(* Logix 5000 project; controller WWTP_SOLIDS_CLX vendor 1 type 14 code 54 rev 17.2; software revision 17.00; part 3 of 16 *)
(* tags used below, declared in another part *)
   Inp : BOOL;   // Alarm Condition Input 1=Alarm
   Cfg_ResetReqd : BOOL;   // 1=Reset required to clear Alarm
   Cfg_AckReqd : BOOL;   // 1=Acknowledge required for Alarm
   Cfg_Severity : SINT;   // 1=Info Only; 2=Warning; 3=Process Exception; 4=Fault
   Cfg_MinDuration : DINT;   // Minimum time (sec) Input must stay on to generate Alarm
   PCmd_Ack : BOOL;   // Program Command to Acknowledge alarm
   PCmd_Inhibit : BOOL;   // Program Command to Inhibit alarm (force Alm to 0)
   PCmd_Uninhibit : BOOL;   // Program Command to Uninhibit alarm
   OCmd_Ack : BOOL;   // Operator Command to Acknowledge alarm
   OCmd_Disable : BOOL;   // Operator Command to Disable alarm (force Alm to 0)
   OCmd_Enable : BOOL;   // Operator Command to Enable alarm
   Alm : BOOL;   // Alarm output 1=In Alarm
   Ack : BOOL;   // Alarm acknowledged status: 1=Ack rcvd
   Disabled : BOOL;   // 1=Alarm has been Disabled by Operator (will not be sent)
   Inhibited : BOOL;   // 1=Alarm has been Inhibited by logic (will not be sent)
   Suppressed : BOOL;   // 1=Alarm has been suppressed (not visible on HMI)
   Rdy_Disable : BOOL;   // Ready to receive OCmd_Disable (enable button)
(* P_Alarm, continued *)

ROUTINE Prescan   (* ladder *)
// Clear "lurking" Commands
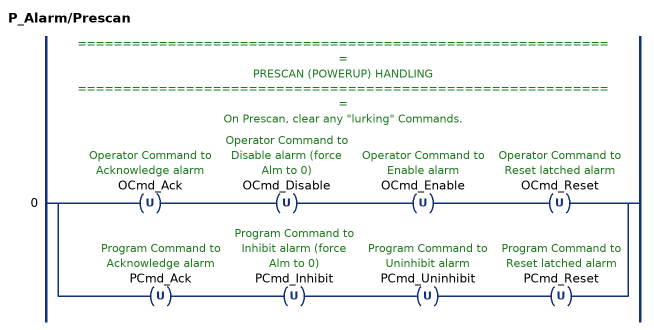
   // ============================================================
   // PRESCAN (POWERUP) HANDLING
   // ============================================================
   // On Prescan, clear any "lurking" Commands.
   0: [OTU(OCmd_Ack) OTU(OCmd_Disable) OTU(OCmd_Enable) OTU(OCmd_Reset) ,OTU(PCmd_Ack) OTU(PCmd_Inhibit) OTU(PCmd_Uninhibit) OTU(PCmd_Reset) ];
END_ROUTINE
END_ADD_ON_INSTRUCTION

ADD_ON_INSTRUCTION P_DIn   (* revision 0.29, ExecutePrescan, ExecuteEnableInFalse *)
// Discrete Input
// Revision note:
// Aligned name, description and local STRING values, sizes, across instructions.
// Help:
// This instruction monitors a discrete (1 / 0) input and checks for alarm conditions.
// The Inp_Gate input must be set (=1, its default value) and the alarm enabled for
// the alarm (Alm) to occur.  The alarm will not occur until the Inp_Gate input has
// been set for the Gate Delay (Cfg_GateDly) time.  The Gate is used to enable the
// alarm when some other condition is true; for example, a high vibration switch should
// only generate an alarm when the associated motor has been running long enough
// to stabilize.
// The alarm is generated when the Inp_PV (process variable) input is different from
// the Inp_Target (target) input.  The Target indicates the "normal" condition.  For
// example, a flow switch should indicate flow when a pump is running and should
// not indicate flow when a pump is stopped.  The pump run status is used as the
// Target input, and when the switch does not match the target (within the allotted
// time), the Alarm (Flow Loss / Switch Failure) is generated.
// NOTE: the Inp_PV is inverted when the rung condition is false -- this allows the
// input to be a condition on the rung with P_DIn rather than mapped into Inp_PV.
// See P_DIn documentation for details.
// This instruction includes a substitute PV capability for a manually-entered state.
// This may be useful when a sensor is out for repair or for simulation and testing.
VAR_INPUT
   Inp_PV : BOOL := 1; {visible}   // Input Signal (process variable) from Sensor
   Inp_PVBad : BOOL;   // Input Comm Status or Quality 1=Bad, 0=OK
   Inp_Target : BOOL := 1; {visible}   // Target State of Input (Alarm if not in Target State)
   Inp_Gate : BOOL := 1; {visible}   // Gate Condition (=1 to enable Alarm)
   Inp_Sim : BOOL;   // 1=Use simulated PV (Set_SimPV); 0=Use Input (Inp_PV)
   Inp_Reset : BOOL;   // 1=Reset Alarm requiring reset
   Cfg_NoSubstPV : BOOL;   // 1=Disallow selection of Substitute PV
   Cfg_NormTextVis : BOOL := 1;   // 1=Display state text in "normal" state (= target), 0=hide (some HMI objects)
   Cfg_PCmdClear : BOOL := 1;   // 1=Clear Program Commands on receipt 0=Leave Set
   Cfg_HasTgtDisagreeAlm : BOOL;   // 1=Target Disagree Alarm exists and will be checked
   Cfg_TgtDisagreeResetReqd : BOOL;   // 1=Target Disagree Alarm is latched in, requires Reset Command to clear
   Cfg_TgtDisagreeAckReqd : BOOL := 1;   // 1=Target Disagree Alarm must be acknowledged
   Cfg_TgtDisagreeSeverity : SINT := 3;   // Target Disagree Alarm Severity: 1=info, 2=warn, 3=excep, 4=fault
   Cfg_GateDly : DINT;   // Time Inp_Gate must be true before Alarm is checked (sec)
   Cfg_Debounce : REAL;   // Minimum time Status must maintain state, (sec)
   Cfg_TgtDisagreeMinDuration : DINT;   // Minimum time Input must disagree with target to generate an Alarm (sec)
   MSet_SubstPV : BOOL;   // Maintenance-Entered Substitute PV
   Set_SimPV : BOOL;   // PV used in Simulation (Inp_Sim=1)
   PCmd_Reset : BOOL;   // Program Command to Reset all latched Alarms
   PCmd_TgtDisagreeAck : BOOL;   // Program Command to Acknowledge the Target Disagree Alarm
   PCmd_TgtDisagreeInhibit : BOOL;   // Program Command to Inhibit the Target Disagree Alarm
   PCmd_TgtDisagreeUninhibit : BOOL;   // Program Command to Uninhibit the Target Disagree Alarm
   MCmd_SubstPV : BOOL;   // Maintenance Command to use Substitute PV (override input)
   MCmd_InpPV : BOOL;   // Maintenance Command to use Input PV (normal)
   OCmd_Reset : BOOL;   // Operator Command to Reset all latched Alarms
END_VAR
VAR_OUTPUT
   Val_Notify : SINT;   // Current Alarm Level and Acknowledgement (enumeration)
   Sts : BOOL; {visible}   // Discrete Input Status (incl. Debounce, Manual Override, if used)
   Sts_PV : BOOL; {visible}   // Discrete Input Status (actual, not subject to Override)
   Sts_SubstPV : BOOL;   // 1=Using Substitute PV (Input being overridden)
   Sts_InpPV : BOOL;   // 1=Using Input PV (normal)
   Sts_PVBad : BOOL;   // Input Comm Status/ Quality (0=OK, 1=Bad)
   Sts_Err : BOOL; {visible}   // 1=Error in Config: see detail bits for reason
   Err_Timer : BOOL;   // 1=Error in Config: Invalid Timer Preset (use 0 to 2147483)
   Err_Alarm : BOOL;   // 1=Error in Config: Invalid Alarm Min Duration or Severity
   Sts_TgtDisagree : BOOL;   // 1=Input is not in Target state
   Alm_TgtDisagree : BOOL;   // 1=Alarm: Input is not in Target state
   Ack_TgtDisagree : BOOL;   // 1=Target Disagree Alarm has been acknowledged
   Sts_TgtDisagreeDisabled : BOOL;   // 1=Target Disagree Alarm is Disabled (not saved or sent)
   Sts_TgtDisagreeInhibited : BOOL;   // 1=Target Disagree Alarm is Inhibited by logic
   Sts_TgtDisagreeSuppressed : BOOL;   // 1=Target Disagree Alarm is Suppressed (logged only)
   Rdy_SubstPV : BOOL;   // 1=Ready for MCmd_SubstPV
   Rdy_InpPV : BOOL;   // 1=Ready for MCmd_InpPV
   Rdy_Reset : BOOL;   // 1=Ready for Operator Alarm Reset Command
END_VAR
VAR
   Wrk_GateDlyT : TIMER;   // Gate Delay timer
   Cfg_Tag : STRING_20 := 'P_DIn';   // Tagname for display on HMI
   Cfg_Desc : STRING_40 := 'Discrete Input';   // Description for display on HMI
   Cfg_Label : STRING_20 := 'Discrete Input';   // Label for graphic symbol displayed on HMI
   Wrk_Sts : BOOL;   // Internal Status (after Manual Override selection)
   TgtDisagree : P_Alarm := (Inp := 1, Cfg_AckReqd := 1, Cfg_Severity := 3, Ack := 1, Rdy_Disable := 1);   // Target Disagree Alarm
   Wrk_FallT : TIMER;   // Timer to ensure Status LOW time on falling edge
   Wrk_RiseT : TIMER;   // Timer to ensure Status HIGH time on rising edge
   Wrk_SubstPV : BOOL;   // Internal flag: Using Substitute PV
   Cfg_1StText : STRING_8 := 'On';   // Text to display in PV=1 State
   Cfg_0StText : STRING_8 := 'Off';   // Text to display in PV=0 State
END_VAR

ROUTINE EnableInFalse   (* ladder *)
// Inverts Inp_PV to allow mapping input using XIC/XIO on rung
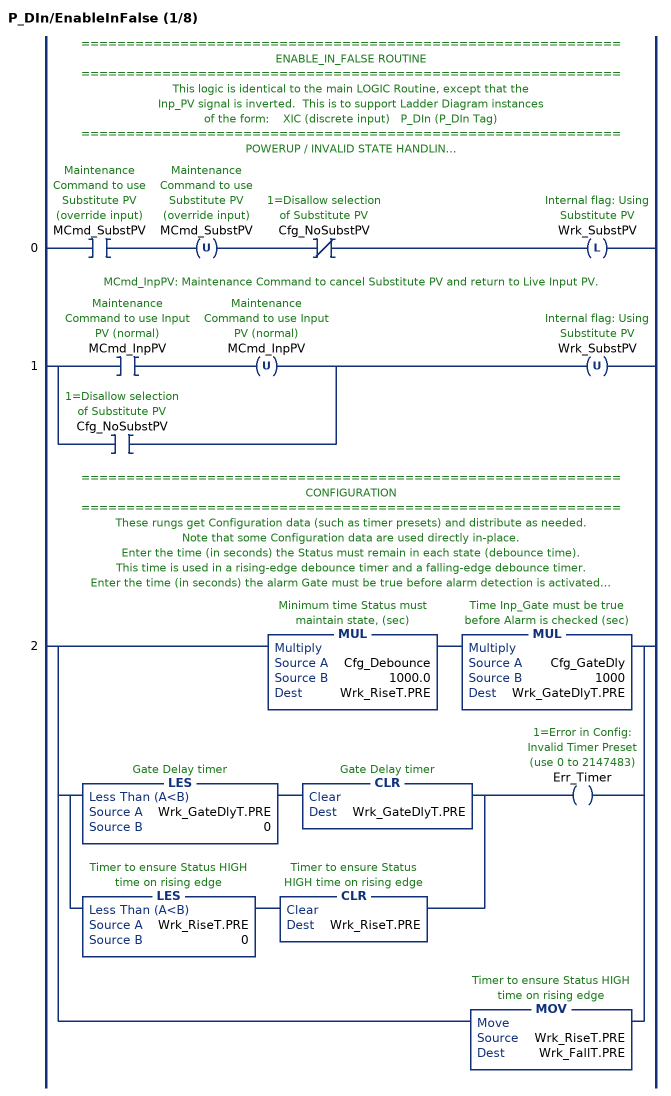
   // ============================================================
   // ENABLE_IN_FALSE ROUTINE
   // ============================================================
   // This logic is identical to the main LOGIC Routine, except that the
   // Inp_PV signal is inverted.  This is to support Ladder Diagram instances
   // of the form:    XIC (discrete input)   P_DIn (P_DIn Tag)
   // ============================================================
   // POWERUP / INVALID STATE HANDLING
   // ============================================================
   // All internal Work (state) bits maintain states through a power cycle and are
   // independent.  No Powerup / Invalid State Handling logic is required.
   // ============================================================
   // COMMAND PROCESSING
   // ============================================================
   // These rungs handle received Commands:
   // NOTE:  Operator Commands for P_Alarm are sent directly to the contained P_Alarm AOI.
   // MCmd_SubstPV: Maintenance Command to select Maintenance-entered substitute PV
   // Do not allow this Commands if Cfg_NoSubstPV is set.
   0: XIC(MCmd_SubstPV)OTU(MCmd_SubstPV)XIO(Cfg_NoSubstPV)OTL(Wrk_SubstPV);
   // MCmd_InpPV: Maintenance Command to cancel Substitute PV and return to Live Input PV.
   1: [XIC(MCmd_InpPV) OTU(MCmd_InpPV) ,XIC(Cfg_NoSubstPV) ]OTU(Wrk_SubstPV);
   // ============================================================
   // CONFIGURATION
   // ============================================================
   // These rungs get Configuration data (such as timer presets) and distribute as needed.
   // Note that some Configuration data are used directly in-place.
   // Enter the time (in seconds) the Status must remain in each state (debounce time).
   // This time is used in a rising-edge debounce timer and a falling-edge debounce timer.
   // Enter the time (in seconds) the alarm Gate must be true before alarm detection is activated.
   // If the timer preset calcuated wraps negative (more than 2.14... million seconds), then establish
   // a valid limit value for the Preset.  Note that a negative timer preset will fault the controller!!!
   2: [MUL(Cfg_Debounce,1000.0,Wrk_RiseT.PRE) MUL(Cfg_GateDly,1000,Wrk_GateDlyT.PRE) ,[LES(Wrk_GateDlyT.PRE,0) CLR(Wrk_GateDlyT.PRE) ,LES(Wrk_RiseT.PRE,0) CLR(Wrk_RiseT.PRE) ] OTE(Err_Timer) ,MOV(Wrk_RiseT.PRE,Wrk_FallT.PRE) ];
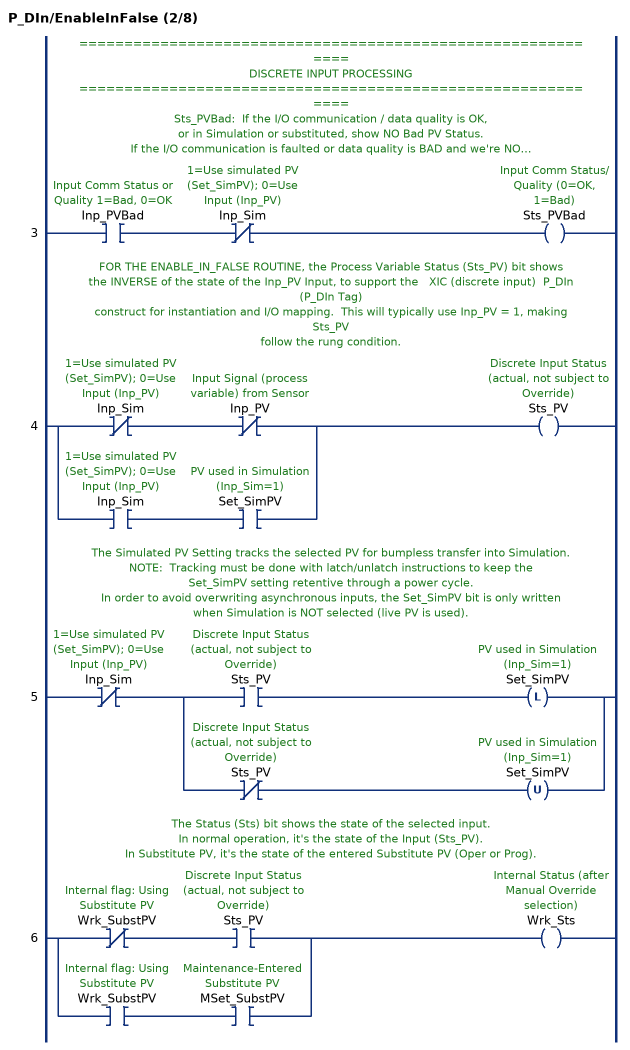
   // ============================================================
   // DISCRETE INPUT PROCESSING
   // ============================================================
   // Sts_PVBad:  If the I/O communication / data quality is OK,
   // or in Simulation or substituted, show NO Bad PV Status.
   // If the I/O communication is faulted or data quality is BAD and we're NOT
   // in Simulation or using substitute PV, show the Bad PV Status.
   3: XIC(Inp_PVBad)XIO(Inp_Sim)OTE(Sts_PVBad);
   // FOR THE ENABLE_IN_FALSE ROUTINE, the Process Variable Status (Sts_PV) bit shows
   // the INVERSE of the state of the Inp_PV Input, to support the   XIC (discrete input)  P_DIn (P_DIn Tag)
   // construct for instantiation and I/O mapping.  This will typically use Inp_PV = 1, making Sts_PV
   // follow the rung condition.
   4: [XIO(Inp_Sim) XIO(Inp_PV) ,XIC(Inp_Sim) XIC(Set_SimPV) ]OTE(Sts_PV);
   // The Simulated PV Setting tracks the selected PV for bumpless transfer into Simulation.
   // NOTE:  Tracking must be done with latch/unlatch instructions to keep the
   // Set_SimPV setting retentive through a power cycle.
   // In order to avoid overwriting asynchronous inputs, the Set_SimPV bit is only written
   // when Simulation is NOT selected (live PV is used).
   5: XIO(Inp_Sim)[XIC(Sts_PV) OTL(Set_SimPV) ,XIO(Sts_PV) OTU(Set_SimPV) ];
   // The Status (Sts) bit shows the state of the selected input.
   // In normal operation, it's the state of the Input (Sts_PV).
   // In Substitute PV, it's the state of the entered Substitute PV (Oper or Prog).
   6: [XIO(Wrk_SubstPV) XIC(Sts_PV) ,XIC(Wrk_SubstPV) XIC(MSet_SubstPV) ]OTE(Wrk_Sts);
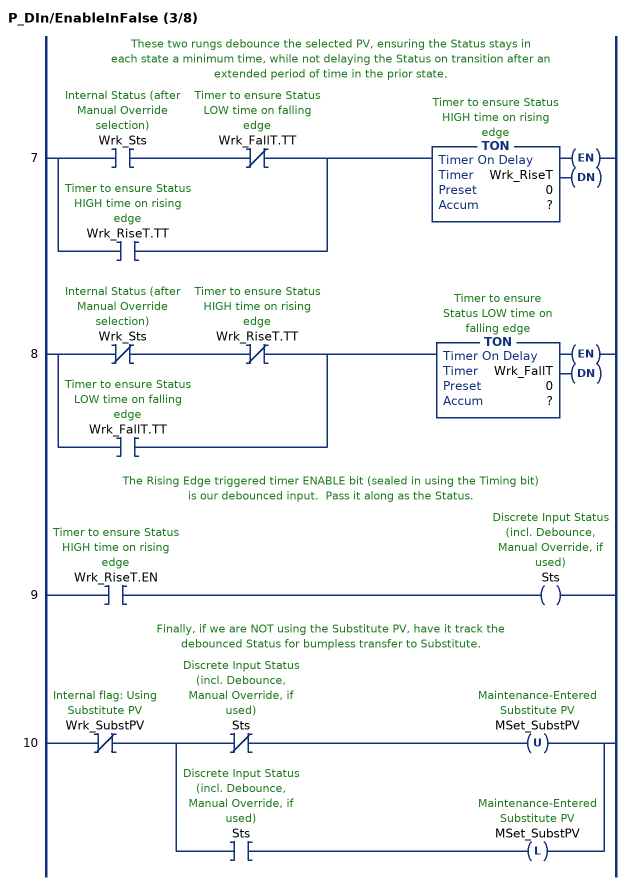
   // These two rungs debounce the selected PV, ensuring the Status stays in
   // each state a minimum time, while not delaying the Status on transition after an
   // extended period of time in the prior state.
   7: [XIC(Wrk_Sts) XIO(Wrk_FallT.TT) ,XIC(Wrk_RiseT.TT) ]TON(Wrk_RiseT,?,?);
   8: [XIO(Wrk_Sts) XIO(Wrk_RiseT.TT) ,XIC(Wrk_FallT.TT) ]TON(Wrk_FallT,?,?);
   // The Rising Edge triggered timer ENABLE bit (sealed in using the Timing bit)
   // is our debounced input.  Pass it along as the Status.
   9: XIC(Wrk_RiseT.EN)OTE(Sts);
   // Finally, if we are NOT using the Substitute PV, have it track the
   // debounced Status for bumpless transfer to Substitute.
   10: XIO(Wrk_SubstPV)[XIO(Sts) OTU(MSet_SubstPV) ,XIC(Sts) OTL(MSet_SubstPV) ];
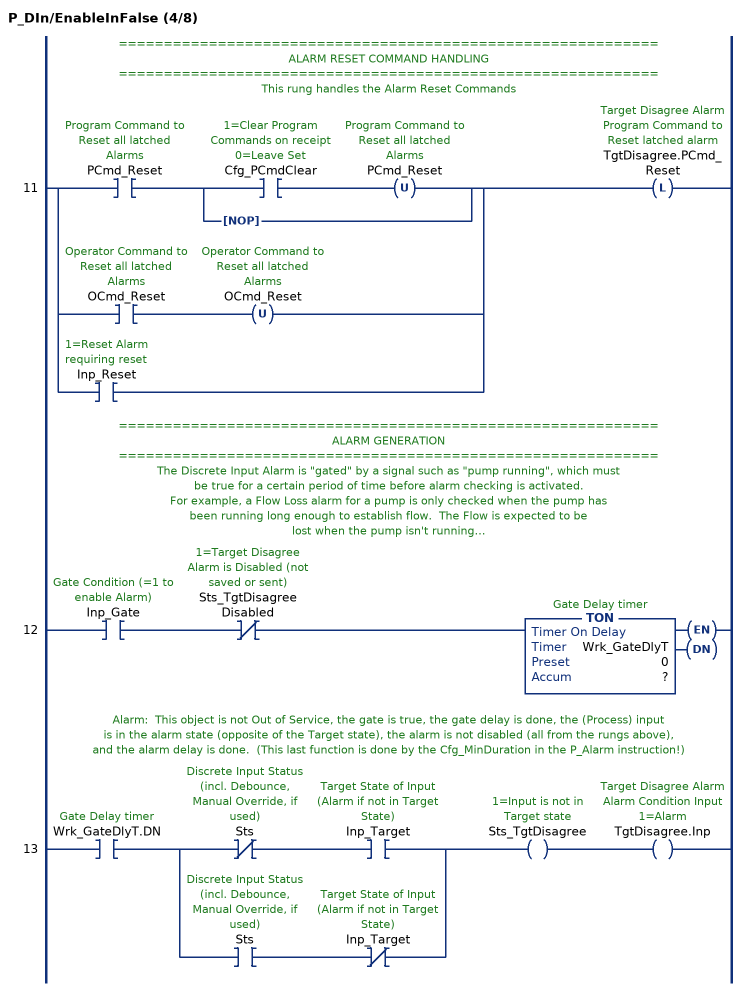
   // ============================================================
   // ALARM RESET COMMAND HANDLING
   // ============================================================
   // This rung handles the Alarm Reset Commands
   11: [XIC(PCmd_Reset) [XIC(Cfg_PCmdClear) OTU(PCmd_Reset) ,NOP() ] ,XIC(OCmd_Reset) OTU(OCmd_Reset) ,XIC(Inp_Reset) ]OTL(TgtDisagree.PCmd_Reset);
   // ============================================================
   // ALARM GENERATION
   // ============================================================
   // The Discrete Input Alarm is "gated" by a signal such as "pump running", which must
   // be true for a certain period of time before alarm checking is activated.
   // For example, a Flow Loss alarm for a pump is only checked when the pump has
   // been running long enough to establish flow.  The Flow is expected to be
   // lost when the pump isn't running!
   // If no gating signal is available, set Inp_Gate to 1 and Cfg_GateT to 0.
   12: XIC(Inp_Gate)XIO(Sts_TgtDisagreeDisabled)TON(Wrk_GateDlyT,?,?);
   // Alarm:  This object is not Out of Service, the gate is true, the gate delay is done, the (Process) input
   // is in the alarm state (opposite of the Target state), the alarm is not disabled (all from the rungs above),
   // and the alarm delay is done.  (This last function is done by the Cfg_MinDuration in the P_Alarm instruction!)
   13: XIC(Wrk_GateDlyT.DN)[XIO(Sts) XIC(Inp_Target) ,XIC(Sts) XIO(Inp_Target) ]OTE(Sts_TgtDisagree)OTE(TgtDisagree.Inp);
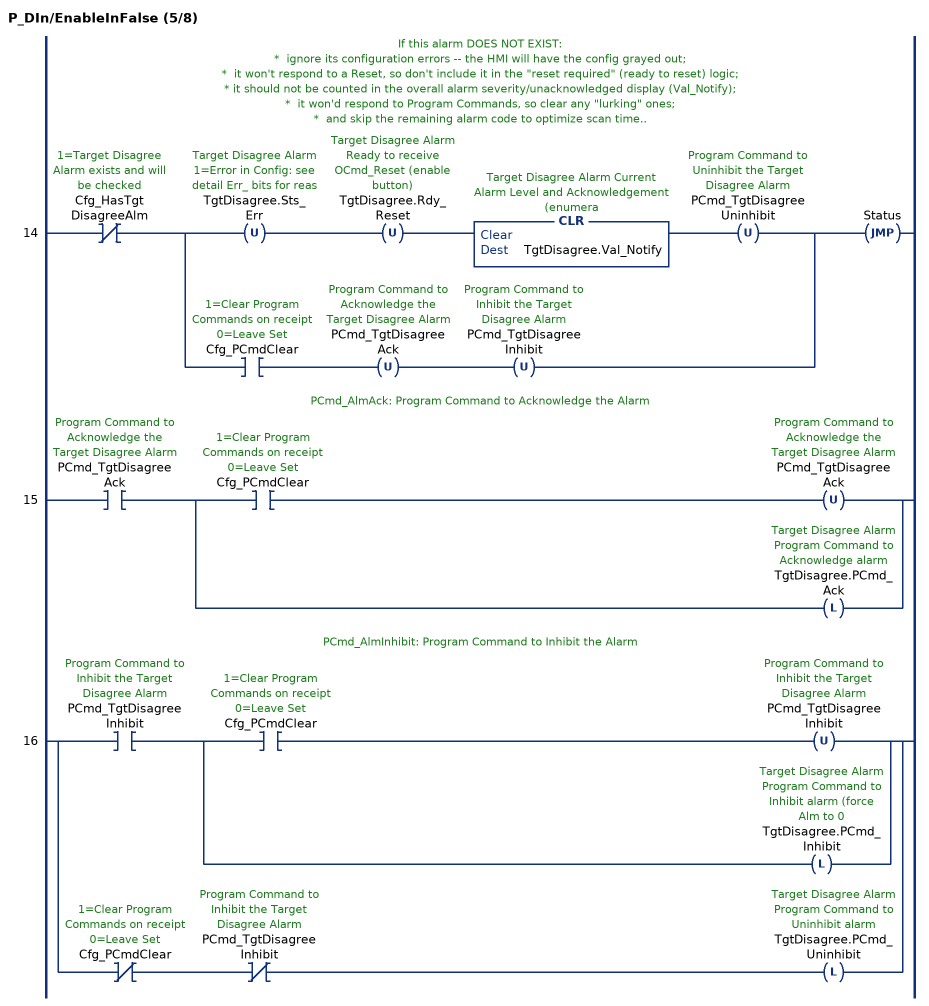
   // If this alarm DOES NOT EXIST:
   // *  ignore its configuration errors -- the HMI will have the config grayed out;
   // *  it won't respond to a Reset, so don't include it in the "reset required" (ready to reset) logic;
   // * it should not be counted in the overall alarm severity/unacknowledged display (Val_Notify);
   // *  it won'd respond to Program Commands, so clear any "lurking" ones;
   // *  and skip the remaining alarm code to optimize scan time..
   14: XIO(Cfg_HasTgtDisagreeAlm)[OTU(TgtDisagree.Sts_Err) OTU(TgtDisagree.Rdy_Reset) CLR(TgtDisagree.Val_Notify) OTU(PCmd_TgtDisagreeUninhibit) ,XIC(Cfg_PCmdClear) OTU(PCmd_TgtDisagreeAck) OTU(PCmd_TgtDisagreeInhibit) ]JMP(Status);
   // PCmd_AlmAck: Program Command to Acknowledge the Alarm
   15: XIC(PCmd_TgtDisagreeAck)[XIC(Cfg_PCmdClear) OTU(PCmd_TgtDisagreeAck) ,OTL(TgtDisagree.PCmd_Ack) ];
   // PCmd_AlmInhibit: Program Command to Inhibit the Alarm
   16: [XIC(PCmd_TgtDisagreeInhibit) [XIC(Cfg_PCmdClear) OTU(PCmd_TgtDisagreeInhibit) ,OTL(TgtDisagree.PCmd_Inhibit) ] ,XIO(Cfg_PCmdClear) XIO(PCmd_TgtDisagreeInhibit) OTL(TgtDisagree.PCmd_Uninhibit) ];
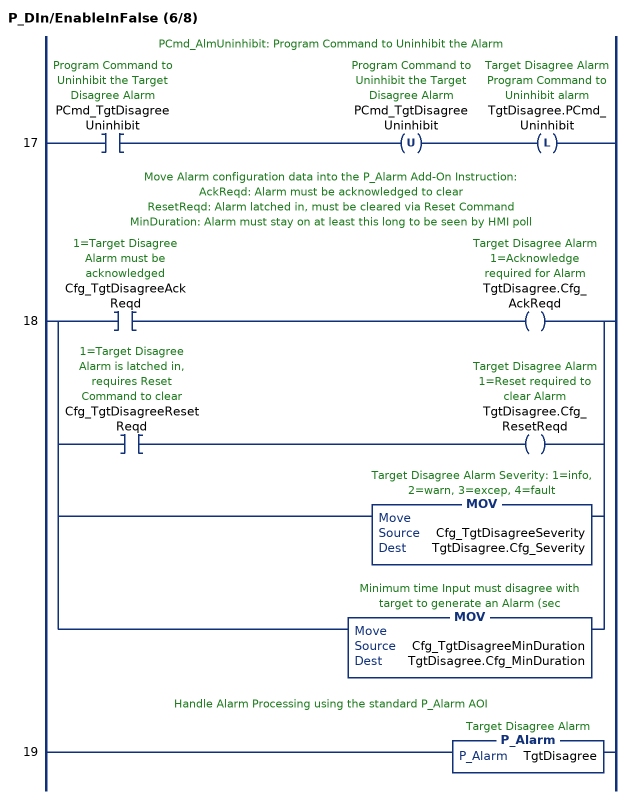
   // PCmd_AlmUninhibit: Program Command to Uninhibit the Alarm
   17: XIC(PCmd_TgtDisagreeUninhibit)OTU(PCmd_TgtDisagreeUninhibit)OTL(TgtDisagree.PCmd_Uninhibit);
   // Move Alarm configuration data into the P_Alarm Add-On Instruction:
   // AckReqd: Alarm must be acknowledged to clear
   // ResetReqd: Alarm latched in, must be cleared via Reset Command
   // MinDuration: Alarm must stay on at least this long to be seen by HMI poll
   18: [XIC(Cfg_TgtDisagreeAckReqd) OTE(TgtDisagree.Cfg_AckReqd) ,XIC(Cfg_TgtDisagreeResetReqd) OTE(TgtDisagree.Cfg_ResetReqd) ,MOV(Cfg_TgtDisagreeSeverity,TgtDisagree.Cfg_Severity) ,MOV(Cfg_TgtDisagreeMinDuration,TgtDisagree.Cfg_MinDuration) ];
   // Handle Alarm Processing using the standard P_Alarm AOI
   19: P_Alarm(TgtDisagree);
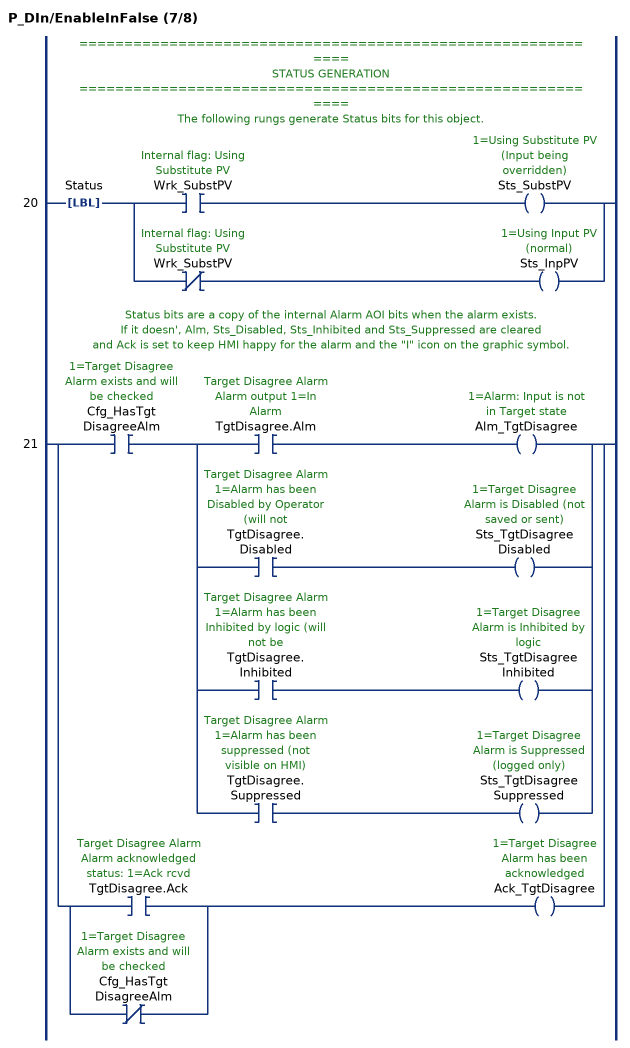
   // ============================================================
   // STATUS GENERATION
   // ============================================================
   // The following rungs generate Status bits for this object.
   20: LBL(Status)[XIC(Wrk_SubstPV) OTE(Sts_SubstPV) ,XIO(Wrk_SubstPV) OTE(Sts_InpPV) ];
   // Status bits are a copy of the internal Alarm AOI bits when the alarm exists.
   // If it doesn', Alm, Sts_Disabled, Sts_Inhibited and Sts_Suppressed are cleared
   // and Ack is set to keep HMI happy for the alarm and the "I" icon on the graphic symbol.
   21: [XIC(Cfg_HasTgtDisagreeAlm) [XIC(TgtDisagree.Alm) OTE(Alm_TgtDisagree) ,XIC(TgtDisagree.Disabled) OTE(Sts_TgtDisagreeDisabled) ,XIC(TgtDisagree.Inhibited) OTE(Sts_TgtDisagreeInhibited) ,XIC(TgtDisagree.Suppressed) OTE(Sts_TgtDisagreeSuppressed) ] ,[XIC(TgtDisagree.Ack) ,XIO(Cfg_HasTgtDisagreeAlm) ] OTE(Ack_TgtDisagree) ];
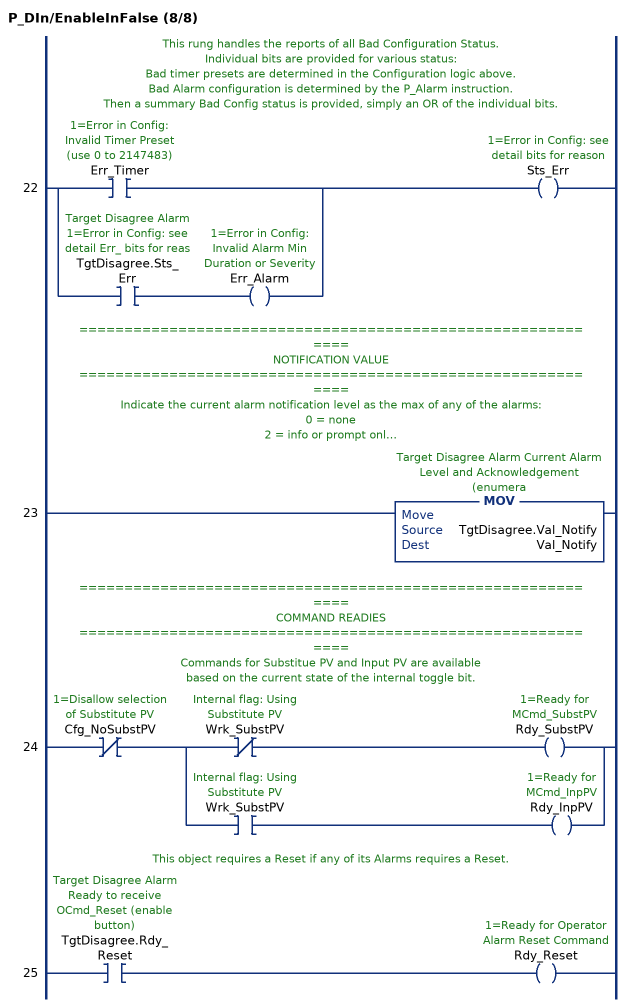
   // This rung handles the reports of all Bad Configuration Status.
   // Individual bits are provided for various status:
   // Bad timer presets are determined in the Configuration logic above.
   // Bad Alarm configuration is determined by the P_Alarm instruction.
   // Then a summary Bad Config status is provided, simply an OR of the individual bits.
   22: [XIC(Err_Timer) ,XIC(TgtDisagree.Sts_Err) OTE(Err_Alarm) ]OTE(Sts_Err);
   // ============================================================
   // NOTIFICATION VALUE
   // ============================================================
   // Indicate the current alarm notification level as the max of any of the alarms:
   // 0 = none
   // 2 = info or prompt only
   // 4 = warning
   // 6 = exception (equipment impact)
   // 8 = fault (equipment failure)
   // Add one for any unsuppressed alarm that is not acknowledged (for blink).
   23: MOV(TgtDisagree.Val_Notify,Val_Notify);
   // ============================================================
   // COMMAND READIES
   // ============================================================
   // Commands for Substitue PV and Input PV are available
   // based on the current state of the internal toggle bit.
   24: XIO(Cfg_NoSubstPV)[XIO(Wrk_SubstPV) OTE(Rdy_SubstPV) ,XIC(Wrk_SubstPV) OTE(Rdy_InpPV) ];
   // This object requires a Reset if any of its Alarms requires a Reset.
   25: XIC(TgtDisagree.Rdy_Reset)OTE(Rdy_Reset);
END_ROUTINE

ROUTINE Logic   (* ladder *)
// Normal Scan - status is updated and alarms are generated
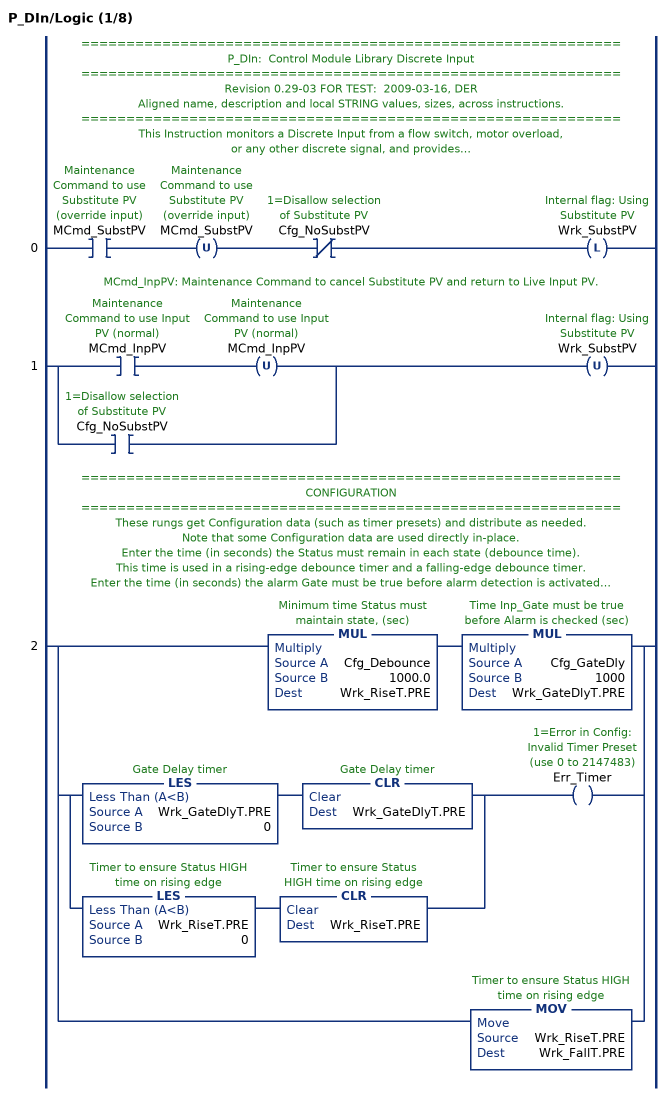
   // ============================================================
   // P_DIn:  Control Module Library Discrete Input
   // ============================================================
   // Revision 0.29-03 FOR TEST:  2009-03-16, DER
   // Aligned name, description and local STRING values, sizes, across instructions.
   // ============================================================
   // This Instruction monitors a Discrete Input from a flow switch, motor overload,
   // or any other discrete signal, and provides:
   // *  Status, with configurable names for the 0- and 1-states
   // *  An Alarm "Gate" signal (with delay), used to enable an Alarm under appropriate process conditions
   // *  A "Target" input -- the Alarm is raised when the input is not in the same
   // state as the Target for a configurable period of time
   // * Input debounce for both the rising and falling transitions
   // * Commands to inhibit or enable alarms
   // * Monitoring of input communication status
   // * Setting of a simulated input signal for process simulation
   // * Selection of Substitute PV (by Maintenance personnel) or normal PV
   // ============================================================
   // POWERUP / INVALID STATE HANDLING
   // ============================================================
   // All internal Work (state) bits maintain states through a power cycle and are
   // independent.  No Powerup / Invalid State Handling logic is required.
   // ============================================================
   // COMMAND PROCESSING
   // ============================================================
   // These rungs handle received Commands:
   // NOTE:  Operator Commands for P_Alarm are sent directly to the contained AOI.
   // MCmd_SubstPV: Maintenance Command to select Maintenance-entered substitute PV
   // Do not allow this Commands if Cfg_NoSubstPV is set.
   0: XIC(MCmd_SubstPV)OTU(MCmd_SubstPV)XIO(Cfg_NoSubstPV)OTL(Wrk_SubstPV);
   // MCmd_InpPV: Maintenance Command to cancel Substitute PV and return to Live Input PV.
   1: [XIC(MCmd_InpPV) OTU(MCmd_InpPV) ,XIC(Cfg_NoSubstPV) ]OTU(Wrk_SubstPV);
   // ============================================================
   // CONFIGURATION
   // ============================================================
   // These rungs get Configuration data (such as timer presets) and distribute as needed.
   // Note that some Configuration data are used directly in-place.
   // Enter the time (in seconds) the Status must remain in each state (debounce time).
   // This time is used in a rising-edge debounce timer and a falling-edge debounce timer.
   // Enter the time (in seconds) the alarm Gate must be true before alarm detection is activated.
   // If the timer preset calcuated wraps negative (more than 2.14... million seconds), then establish
   // a valid limit value for the Preset.  Note that a negative timer preset will fault the controller!!!
   2: [MUL(Cfg_Debounce,1000.0,Wrk_RiseT.PRE) MUL(Cfg_GateDly,1000,Wrk_GateDlyT.PRE) ,[LES(Wrk_GateDlyT.PRE,0) CLR(Wrk_GateDlyT.PRE) ,LES(Wrk_RiseT.PRE,0) CLR(Wrk_RiseT.PRE) ] OTE(Err_Timer) ,MOV(Wrk_RiseT.PRE,Wrk_FallT.PRE) ];
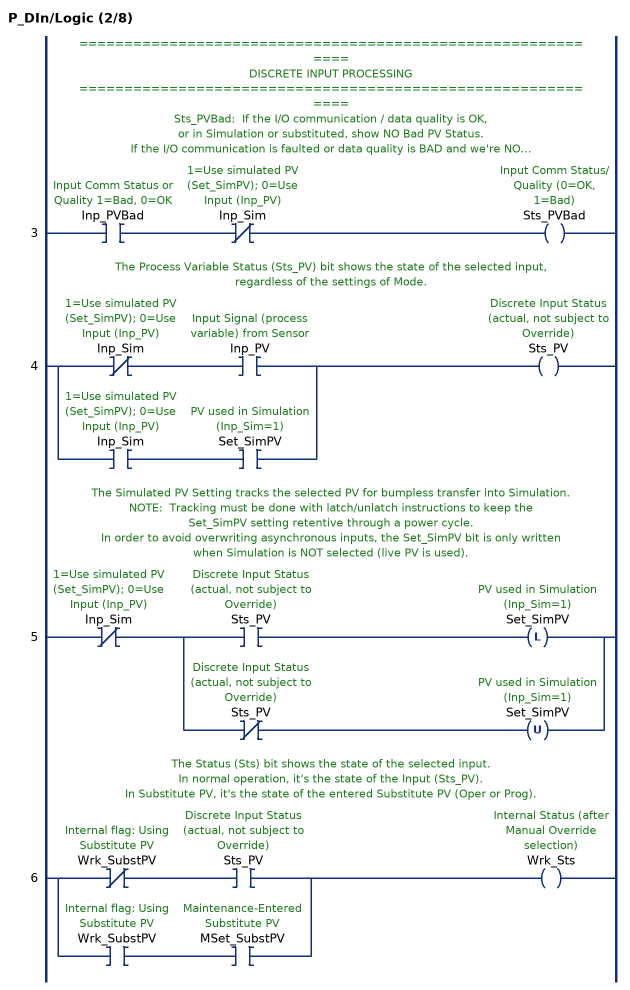
   // ============================================================
   // DISCRETE INPUT PROCESSING
   // ============================================================
   // Sts_PVBad:  If the I/O communication / data quality is OK,
   // or in Simulation or substituted, show NO Bad PV Status.
   // If the I/O communication is faulted or data quality is BAD and we're NOT
   // in Simulation or using substitute PV, show the Bad PV Status.
   3: XIC(Inp_PVBad)XIO(Inp_Sim)OTE(Sts_PVBad);
   // The Process Variable Status (Sts_PV) bit shows the state of the selected input,
   // regardless of the settings of Mode.
   4: [XIO(Inp_Sim) XIC(Inp_PV) ,XIC(Inp_Sim) XIC(Set_SimPV) ]OTE(Sts_PV);
   // The Simulated PV Setting tracks the selected PV for bumpless transfer into Simulation.
   // NOTE:  Tracking must be done with latch/unlatch instructions to keep the
   // Set_SimPV setting retentive through a power cycle.
   // In order to avoid overwriting asynchronous inputs, the Set_SimPV bit is only written
   // when Simulation is NOT selected (live PV is used).
   5: XIO(Inp_Sim)[XIC(Sts_PV) OTL(Set_SimPV) ,XIO(Sts_PV) OTU(Set_SimPV) ];
   // The Status (Sts) bit shows the state of the selected input.
   // In normal operation, it's the state of the Input (Sts_PV).
   // In Substitute PV, it's the state of the entered Substitute PV (Oper or Prog).
   6: [XIO(Wrk_SubstPV) XIC(Sts_PV) ,XIC(Wrk_SubstPV) XIC(MSet_SubstPV) ]OTE(Wrk_Sts);
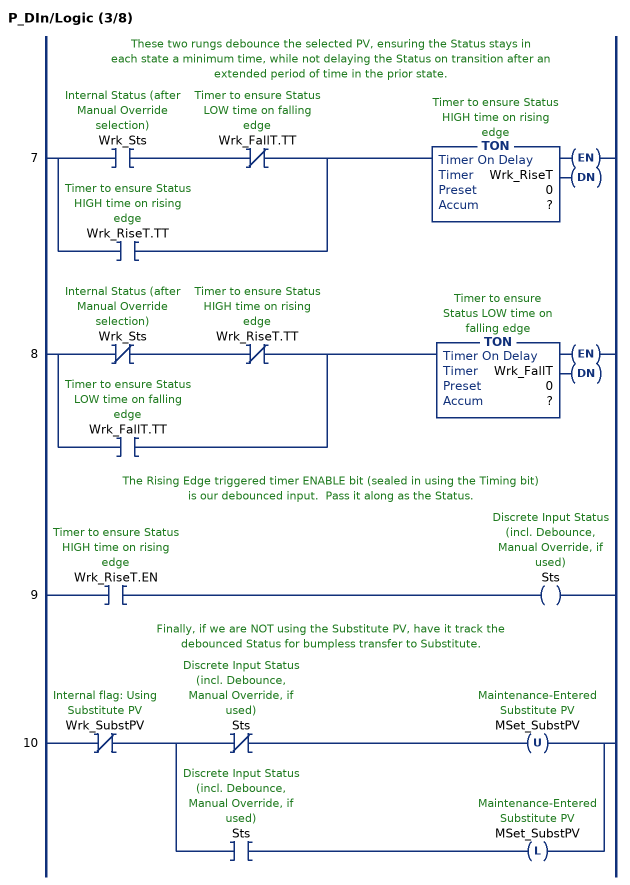
   // These two rungs debounce the selected PV, ensuring the Status stays in
   // each state a minimum time, while not delaying the Status on transition after an
   // extended period of time in the prior state.
   7: [XIC(Wrk_Sts) XIO(Wrk_FallT.TT) ,XIC(Wrk_RiseT.TT) ]TON(Wrk_RiseT,?,?);
   8: [XIO(Wrk_Sts) XIO(Wrk_RiseT.TT) ,XIC(Wrk_FallT.TT) ]TON(Wrk_FallT,?,?);
   // The Rising Edge triggered timer ENABLE bit (sealed in using the Timing bit)
   // is our debounced input.  Pass it along as the Status.
   9: XIC(Wrk_RiseT.EN)OTE(Sts);
   // Finally, if we are NOT using the Substitute PV, have it track the
   // debounced Status for bumpless transfer to Substitute.
   10: XIO(Wrk_SubstPV)[XIO(Sts) OTU(MSet_SubstPV) ,XIC(Sts) OTL(MSet_SubstPV) ];
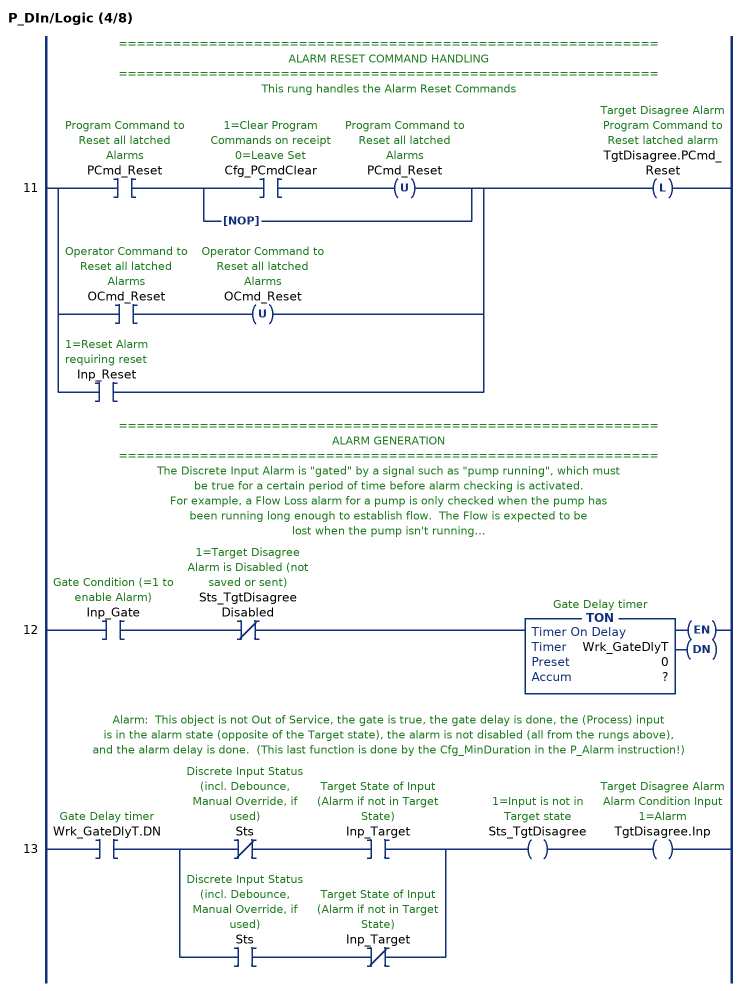
   // ============================================================
   // ALARM RESET COMMAND HANDLING
   // ============================================================
   // This rung handles the Alarm Reset Commands
   11: [XIC(PCmd_Reset) [XIC(Cfg_PCmdClear) OTU(PCmd_Reset) ,NOP() ] ,XIC(OCmd_Reset) OTU(OCmd_Reset) ,XIC(Inp_Reset) ]OTL(TgtDisagree.PCmd_Reset);
   // ============================================================
   // ALARM GENERATION
   // ============================================================
   // The Discrete Input Alarm is "gated" by a signal such as "pump running", which must
   // be true for a certain period of time before alarm checking is activated.
   // For example, a Flow Loss alarm for a pump is only checked when the pump has
   // been running long enough to establish flow.  The Flow is expected to be
   // lost when the pump isn't running!
   // If no gating signal is available, set Inp_Gate to 1 and Cfg_GateT to 0.
   12: XIC(Inp_Gate)XIO(Sts_TgtDisagreeDisabled)TON(Wrk_GateDlyT,?,?);
   // Alarm:  This object is not Out of Service, the gate is true, the gate delay is done, the (Process) input
   // is in the alarm state (opposite of the Target state), the alarm is not disabled (all from the rungs above),
   // and the alarm delay is done.  (This last function is done by the Cfg_MinDuration in the P_Alarm instruction!)
   13: XIC(Wrk_GateDlyT.DN)[XIO(Sts) XIC(Inp_Target) ,XIC(Sts) XIO(Inp_Target) ]OTE(Sts_TgtDisagree)OTE(TgtDisagree.Inp);
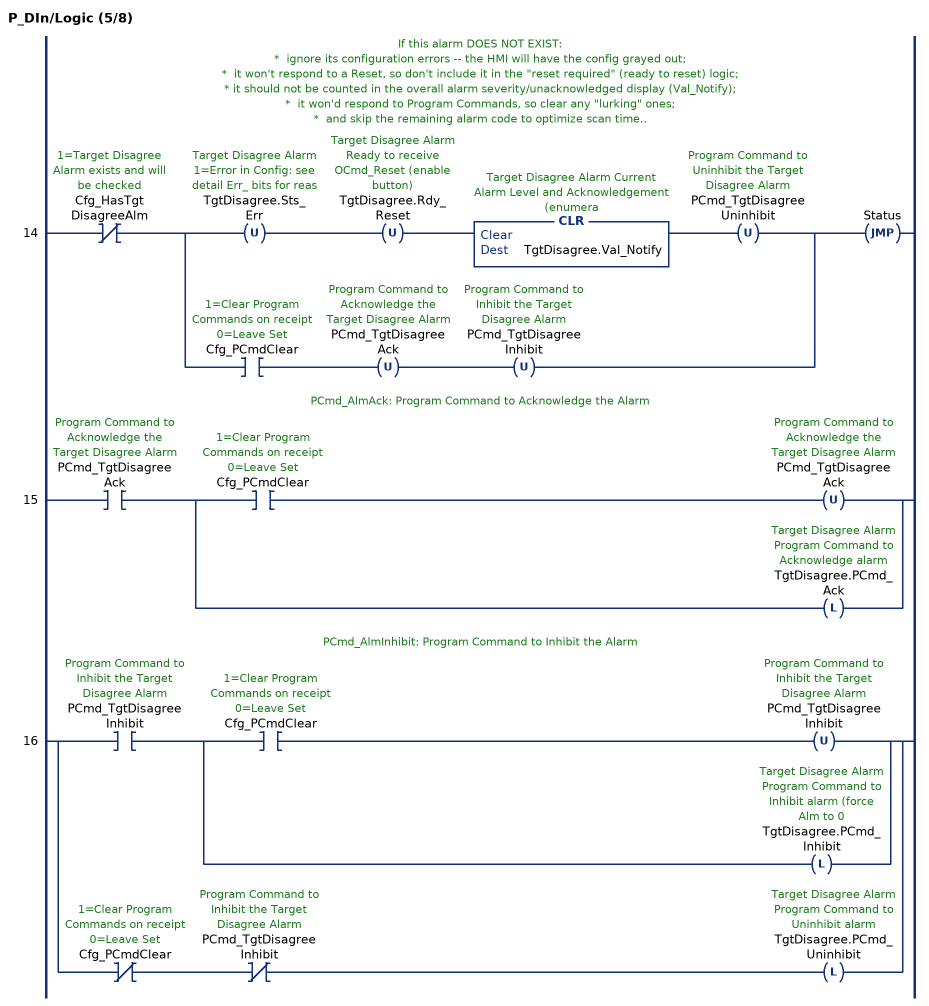
   // If this alarm DOES NOT EXIST:
   // *  ignore its configuration errors -- the HMI will have the config grayed out;
   // *  it won't respond to a Reset, so don't include it in the "reset required" (ready to reset) logic;
   // * it should not be counted in the overall alarm severity/unacknowledged display (Val_Notify);
   // *  it won'd respond to Program Commands, so clear any "lurking" ones;
   // *  and skip the remaining alarm code to optimize scan time..
   14: XIO(Cfg_HasTgtDisagreeAlm)[OTU(TgtDisagree.Sts_Err) OTU(TgtDisagree.Rdy_Reset) CLR(TgtDisagree.Val_Notify) OTU(PCmd_TgtDisagreeUninhibit) ,XIC(Cfg_PCmdClear) OTU(PCmd_TgtDisagreeAck) OTU(PCmd_TgtDisagreeInhibit) ]JMP(Status);
   // PCmd_AlmAck: Program Command to Acknowledge the Alarm
   15: XIC(PCmd_TgtDisagreeAck)[XIC(Cfg_PCmdClear) OTU(PCmd_TgtDisagreeAck) ,OTL(TgtDisagree.PCmd_Ack) ];
   // PCmd_AlmInhibit: Program Command to Inhibit the Alarm
   16: [XIC(PCmd_TgtDisagreeInhibit) [XIC(Cfg_PCmdClear) OTU(PCmd_TgtDisagreeInhibit) ,OTL(TgtDisagree.PCmd_Inhibit) ] ,XIO(Cfg_PCmdClear) XIO(PCmd_TgtDisagreeInhibit) OTL(TgtDisagree.PCmd_Uninhibit) ];
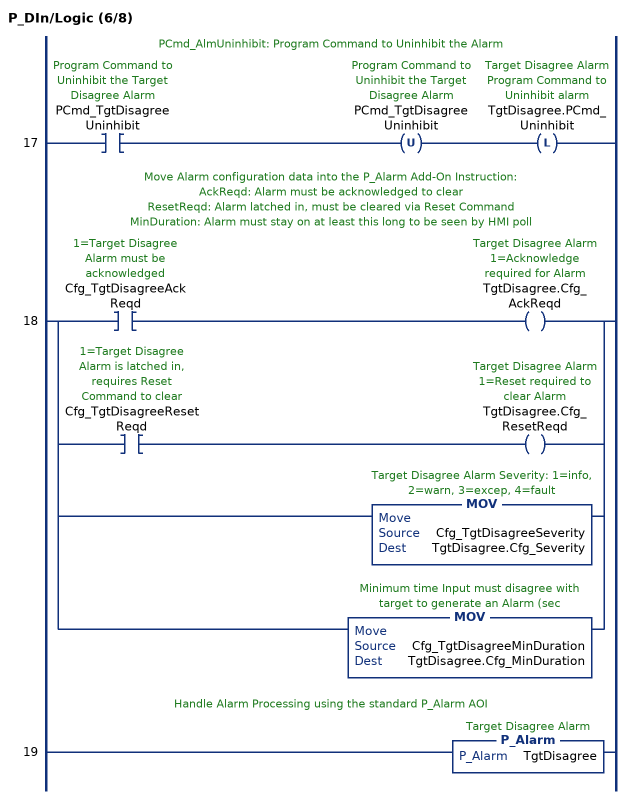
   // PCmd_AlmUninhibit: Program Command to Uninhibit the Alarm
   17: XIC(PCmd_TgtDisagreeUninhibit)OTU(PCmd_TgtDisagreeUninhibit)OTL(TgtDisagree.PCmd_Uninhibit);
   // Move Alarm configuration data into the P_Alarm Add-On Instruction:
   // AckReqd: Alarm must be acknowledged to clear
   // ResetReqd: Alarm latched in, must be cleared via Reset Command
   // MinDuration: Alarm must stay on at least this long to be seen by HMI poll
   18: [XIC(Cfg_TgtDisagreeAckReqd) OTE(TgtDisagree.Cfg_AckReqd) ,XIC(Cfg_TgtDisagreeResetReqd) OTE(TgtDisagree.Cfg_ResetReqd) ,MOV(Cfg_TgtDisagreeSeverity,TgtDisagree.Cfg_Severity) ,MOV(Cfg_TgtDisagreeMinDuration,TgtDisagree.Cfg_MinDuration) ];
   // Handle Alarm Processing using the standard P_Alarm AOI
   19: P_Alarm(TgtDisagree);
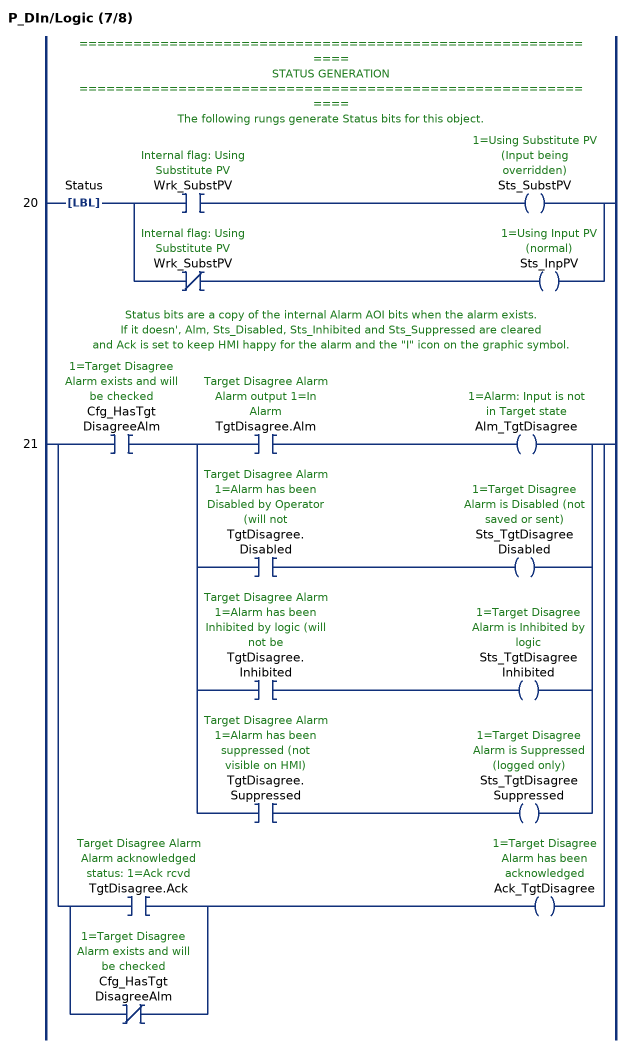
   // ============================================================
   // STATUS GENERATION
   // ============================================================
   // The following rungs generate Status bits for this object.
   20: LBL(Status)[XIC(Wrk_SubstPV) OTE(Sts_SubstPV) ,XIO(Wrk_SubstPV) OTE(Sts_InpPV) ];
   // Status bits are a copy of the internal Alarm AOI bits when the alarm exists.
   // If it doesn', Alm, Sts_Disabled, Sts_Inhibited and Sts_Suppressed are cleared
   // and Ack is set to keep HMI happy for the alarm and the "I" icon on the graphic symbol.
   21: [XIC(Cfg_HasTgtDisagreeAlm) [XIC(TgtDisagree.Alm) OTE(Alm_TgtDisagree) ,XIC(TgtDisagree.Disabled) OTE(Sts_TgtDisagreeDisabled) ,XIC(TgtDisagree.Inhibited) OTE(Sts_TgtDisagreeInhibited) ,XIC(TgtDisagree.Suppressed) OTE(Sts_TgtDisagreeSuppressed) ] ,[XIC(TgtDisagree.Ack) ,XIO(Cfg_HasTgtDisagreeAlm) ] OTE(Ack_TgtDisagree) ];
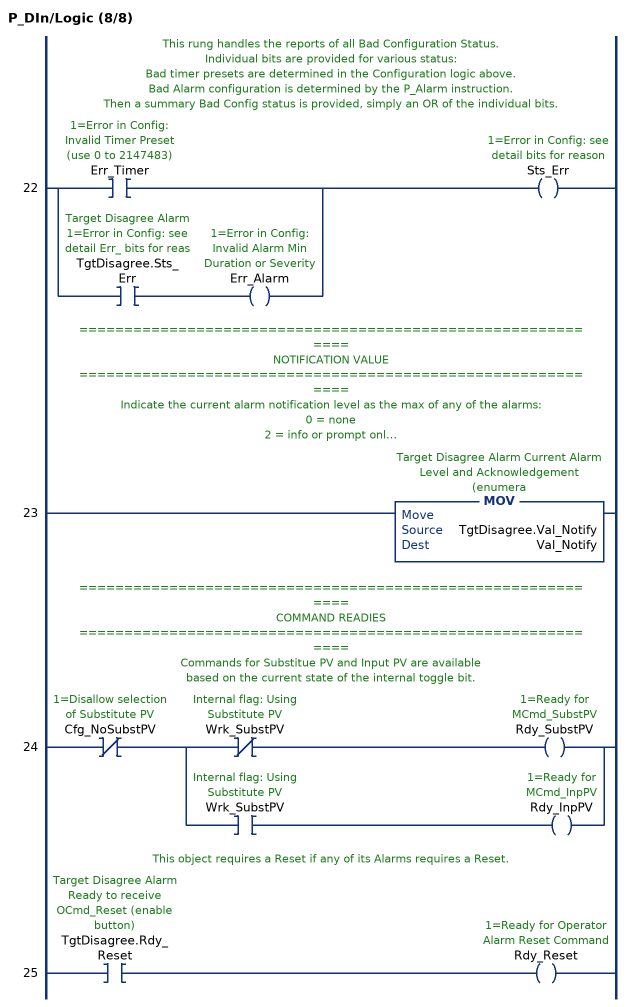
   // This rung handles the reports of all Bad Configuration Status.
   // Individual bits are provided for various status:
   // Bad timer presets are determined in the Configuration logic above.
   // Bad Alarm configuration is determined by the P_Alarm instruction.
   // Then a summary Bad Config status is provided, simply an OR of the individual bits.
   22: [XIC(Err_Timer) ,XIC(TgtDisagree.Sts_Err) OTE(Err_Alarm) ]OTE(Sts_Err);
   // ============================================================
   // NOTIFICATION VALUE
   // ============================================================
   // Indicate the current alarm notification level as the max of any of the alarms:
   // 0 = none
   // 2 = info or prompt only
   // 4 = warning
   // 6 = exception (equipment impact)
   // 8 = fault (equipment failure)
   // Add one for any unsuppressed alarm that is not acknowledged (for blink).
   23: MOV(TgtDisagree.Val_Notify,Val_Notify);
   // ============================================================
   // COMMAND READIES
   // ============================================================
   // Commands for Substitue PV and Input PV are available
   // based on the current state of the internal toggle bit.
   24: XIO(Cfg_NoSubstPV)[XIO(Wrk_SubstPV) OTE(Rdy_SubstPV) ,XIC(Wrk_SubstPV) OTE(Rdy_InpPV) ];
   // This object requires a Reset if any of its Alarms requires a Reset.
   25: XIC(TgtDisagree.Rdy_Reset)OTE(Rdy_Reset);
END_ROUTINE

ROUTINE Prescan   (* ladder *)
// Clear "lurking" Commands
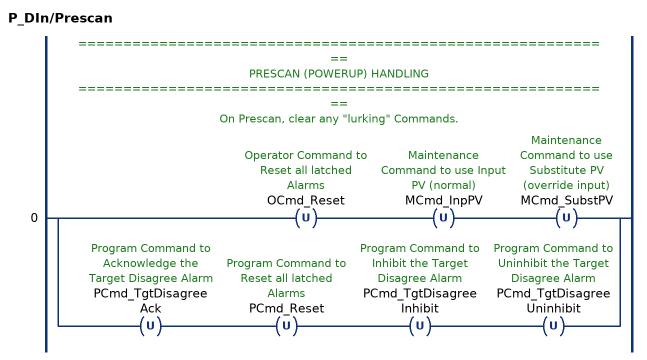
   // ============================================================
   // PRESCAN (POWERUP) HANDLING
   // ============================================================
   // On Prescan, clear any "lurking" Commands.
   0: [OTU(OCmd_Reset) OTU(MCmd_InpPV) OTU(MCmd_SubstPV) ,OTU(PCmd_TgtDisagreeAck) OTU(PCmd_Reset) OTU(PCmd_TgtDisagreeInhibit) OTU(PCmd_TgtDisagreeUninhibit) ];
END_ROUTINE
END_ADD_ON_INSTRUCTION
